INTERFACE I_PropertyVisitor

METHOD VisitProperty
VAR_INPUT
	VisitingProperty : I_Property;
END_VAR
END_METHOD

END_INTERFACE

(* stored: Version 1.1.0.1, ProductVersion 3.1.4024.12
   Itf I_PropertyVisitor: Id {e42b97e1-75a0-0ee6-308b-79206bd66f61}
   Method VisitProperty: Id {c56ceef6-7473-08a2-0bb7-aa4c5609f41d} *)
